FUNCTION_BLOCK Cmd IMPLEMENTS Cyclic
VAR
	startProcess : NT_StartProcess;
END_VAR

{attribute 'monitoring' := 'call'}
PROPERTY Busy : BOOL
GET
Busy := startProcess.BUSY;
END_GET
END_PROPERTY

METHOD Cyclic
startProcess(START := FALSE);
END_METHOD

METHOD Execute
VAR_INPUT
	command : T_MaxString;
	arguments : T_MaxString;
	workingDirectory : T_MaxString;
END_VAR
startProcess(
	DIRNAME := workingDirectory,
	PATHSTR := command,
	COMNDLINE := arguments,
	START := TRUE
);
END_METHOD

END_FUNCTION_BLOCK

(* stored: Version 1.1.0.1
   POU Cmd: Id {e23cdf38-cc76-0c17-2044-3ae4f0301a3a}, SpecialFunc None
   Property Busy: Id {f4f874ce-deca-0e62-3247-4257d5a8c677}
   Get Get: Id {eea6cd53-5635-0863-1b3b-41b5fae984cc}
   Method Cyclic: Id {ed11f2c0-e81a-0565-3a5c-1410b332b0d4}
   Method Execute: Id {351eff9e-be49-0b05-0b20-79f307f3c593} *)
